FUNCTION_BLOCK VACUUM_CONTROL (* Extracted Composite Function Block Type *)
  (* Standard: 61499-2 *)
  (* Version 4/29/2023, Dmitrii *)
  PACKAGE UAO.Hackathon;
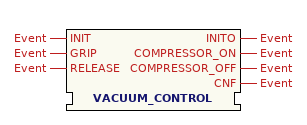
  EVENT_INPUT
    INIT; (* Initializes the symbolic link data source FB with N (1 <= N <= 16) variables *)
    GRIP; (* Grip workpiece *)
    RELEASE; (* Release workpiece *)
  END_EVENT
  EVENT_OUTPUT
    INITO; (* Initialization confirm *)
    COMPRESSOR_ON; (* Request to turn on compressor *)
    COMPRESSOR_OFF; (* Request ot turn off compressor *)
    CNF; (* Vacuum operation confirmation *)
  END_EVENT
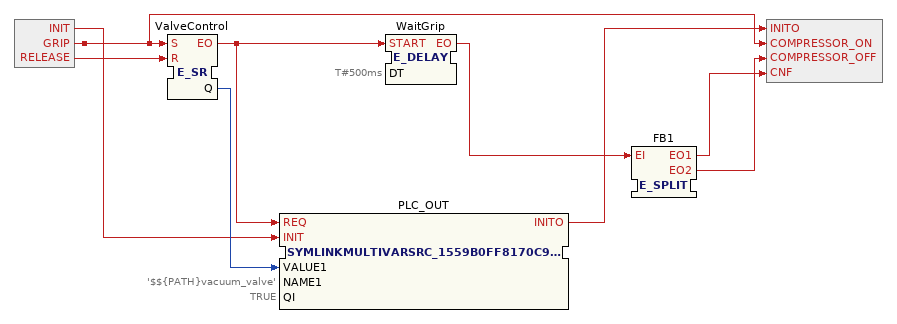
  FBS
    WaitGrip : E_DELAY(DT := T#500ms);
    ValveControl : E_SR;
    PLC_OUT : SYMLINKMULTIVARSRC_1559B0FF8170C9BA0(NAME1 := '$${PATH}vacuum_valve', QI := TRUE); {SET_ATTRIBUTE(Configuration.GenericFBType.InterfaceParams, Runtime.System#I:=1;VALUE${I$}:BOOL)}
    FB1 : E_SPLIT;
  END_FBS
  EVENT_CONNECTIONS
    ValveControl.EO TO WaitGrip.START;
    ValveControl.EO TO PLC_OUT.REQ;
    INIT TO PLC_OUT.INIT;
    PLC_OUT.INITO TO INITO;
    GRIP TO ValveControl.S;
    RELEASE TO ValveControl.R;
    GRIP TO COMPRESSOR_ON;
    WaitGrip.EO TO FB1.EI;
    FB1.EO1 TO CNF;
    FB1.EO2 TO COMPRESSOR_OFF;
  END_CONNECTIONS
  DATA_CONNECTIONS
    ValveControl.Q TO PLC_OUT.VALUE1;
  END_CONNECTIONS
END_FUNCTION_BLOCK
